// TIA Portal V20 export
FUNCTION_BLOCK "FB_Get_In_Rework_Conveyor_Belt"   // FB9, LAD
{ S7_Optimized_Access := 'TRUE' }
// stored: AutoNumber false, MemoryReserve 100, SetENOAutomatically false
   VAR_INPUT
      Emergency_Stop_Release : Bool;
      Start : Bool;
      Sensor_Water_Fountain_Exit_Functional_Test_Spinner_Conveyor_Belt : Bool;
      Sensor_Spinner_Exit_Functional_Test_Position_Withdrawn : Bool;
      Sensor_Spinner_Exit_Functional_Test_Position_Advanced : Bool;
      Sensor_Water_Fountain_Geting_Entrace_Rework_Conveyor_Belt_Start : Bool;
      Sensor_Water_Fountain_Geting_Entrace_Rework_Conveyor_Belt_Finish : Bool;
   END_VAR
   VAR_OUTPUT
      Turn_On_Conveyor_Belt_Motor_Rework_Conveyor_Belt_Get_Exit_Funcional_Test : Bool;
   END_VAR
BEGIN

REGION Network 1
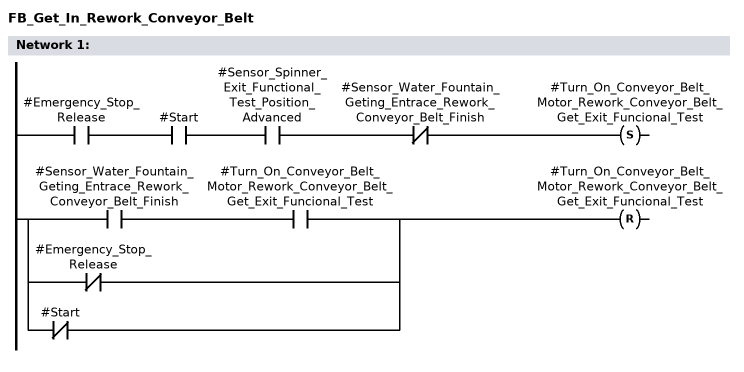
   RUNG wire#powerrail
      Contact( #Emergency_Stop_Release )
      Contact( #Start )
      Contact( #Sensor_Spinner_Exit_Functional_Test_Position_Advanced )
      I_Contact( #Sensor_Water_Fountain_Geting_Entrace_Rework_Conveyor_Belt_Finish )
      S_Coil( #Turn_On_Conveyor_Belt_Motor_Rework_Conveyor_Belt_Get_Exit_Funcional_Test )
   END_RUNG
   RUNG wire#powerrail
      Contact( #Sensor_Water_Fountain_Geting_Entrace_Rework_Conveyor_Belt_Finish )
      Contact( #Turn_On_Conveyor_Belt_Motor_Rework_Conveyor_Belt_Get_Exit_Funcional_Test )
      wire#w1
      R_Coil( #Turn_On_Conveyor_Belt_Motor_Rework_Conveyor_Belt_Get_Exit_Funcional_Test )
   END_RUNG
   RUNG wire#powerrail
      I_Contact( #Emergency_Stop_Release )
   END_RUNG wire#w1
   RUNG wire#powerrail
      I_Contact( #Start )
   END_RUNG wire#w1
   // the same network as SCL:
   IF #Emergency_Stop_Release AND #Start AND #Sensor_Spinner_Exit_Functional_Test_Position_Advanced AND NOT #Sensor_Water_Fountain_Geting_Entrace_Rework_Conveyor_Belt_Finish THEN
       #Turn_On_Conveyor_Belt_Motor_Rework_Conveyor_Belt_Get_Exit_Funcional_Test := TRUE;
   END_IF;
   IF (#Sensor_Water_Fountain_Geting_Entrace_Rework_Conveyor_Belt_Finish AND #Turn_On_Conveyor_Belt_Motor_Rework_Conveyor_Belt_Get_Exit_Funcional_Test) OR NOT #Emergency_Stop_Release OR NOT #Start THEN
       #Turn_On_Conveyor_Belt_Motor_Rework_Conveyor_Belt_Get_Exit_Funcional_Test := FALSE;
   END_IF;
END_REGION
END_FUNCTION_BLOCK
